// Mitsubishi GX Works2 project: CT_PLC_DK_ServoMitsu   PLC: FX1S

PROGRAM MAIN
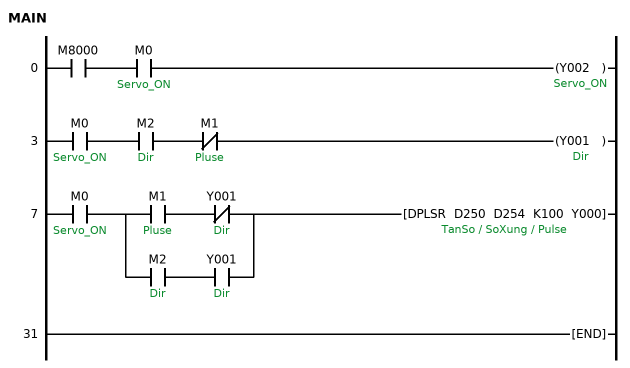
0     LD      M8000
      AND     M0  ; Servo_ON
      OUT     Y002  ; Servo_ON
3     LD      M0  ; Servo_ON
      AND     M2  ; Dir
      ANI     M1  ; Pluse
      OUT     Y001  ; Dir
7     LD      M0  ; Servo_ON
      LD      M1  ; Pluse
      ANI     Y001  ; Dir
      LD      M2  ; Dir
      AND     Y001  ; Dir
      ORB
      ANB
      DPLSR   D250 D254 K100 Y000  ; TanSo / SoXung / Pulse
31    END
END_PROGRAM
